// TIA Portal V19 export
ORGANIZATION_BLOCK "Startup"   // OB100, LAD, Startup
TITLE = "Complete Restart"
// stored: SetENOAutomatically false
   VAR_INPUT
      LostRetentive : Bool;   // True if retentive data are lost
      LostRTC : Bool;   // True if date and time are lost
   END_VAR
BEGIN

REGION Network 1
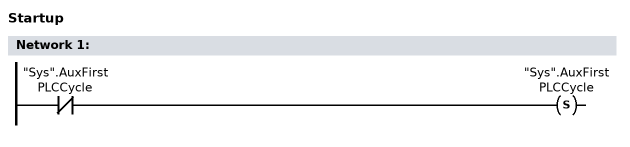
   RUNG wire#powerrail
      I_Contact( "Sys".AuxFirstPLCCycle )
      S_Coil( "Sys".AuxFirstPLCCycle )
   END_RUNG
   // the same network as SCL:
   IF NOT "Sys".AuxFirstPLCCycle THEN "Sys".AuxFirstPLCCycle := TRUE; END_IF;
END_REGION
END_ORGANIZATION_BLOCK
